(* Log/debug/error message fifo *)
FUNCTION_BLOCK FB_LogFifo
VAR_INPUT
	bLog		: BOOL 		:= FALSE;(* TRUE => Enable log message output, FALSE => Disable *)
	sPrefix		: STRING 	:= 'Unknown::';(* Log message description string (allows the identification of log message source) *)
	
	sMessage	: STRING 	:= '';(* String message to add (write) to the fifo *)
	nErrID		: UDINT 	:= 0;(* Error code to add (write) to the fifo *)
	hSocket		: T_HSOCKET;(* Socket connection handle *)
END_VAR
VAR_OUTPUT
	bOk			: BOOL;(* TRUE = New entry added or removed succesfully, FALSE = Fifo overflow or fifo empty *)
	sGet		: T_MaxString := '';(* String entry removed (read) from fifo *)
	nCount		: UDINT := 0;(* Number of fifo entries *)
END_VAR
VAR
	fbBuffer 	: FB_StringRingBuffer;(* Basic (lower level) string buffer control function block *)
	buffer		: ARRAY[0..PLCPRJ_BUFFER_SIZE] OF BYTE;(* Internal buffer memory *)
	sSource		: T_MaxString;	
	sPut		: T_MaxString;
END_VAR

;

ACTION Clear:
(* Clears all fifo entries *)
fbBuffer.A_Reset( 	pBuffer := ADR( buffer ), cbBuffer := SIZEOF( buffer ), 
					bOk=>bOk, nCount=>nCount, getValue=>sGet );
END_ACTION

ACTION Error:
(* Adds new fifo entry *)
IF nErrID = 0 THEN
	sSource := '::Error: 0x';
ELSIF ( nErrID AND 16#80000000) = 16#80000000 THEN
	IF nErrID = 16#80072746 THEN
		sSource := '::Win32 error (the connection is reset by remote side): 0x';
	ELSE
		sSource := '::Win32 error: 0x';
	END_IF
ELSIF (nErrID AND 16#00008100) = 16#00008100 THEN
	CASE nErrID OF
		PLCPRJ_ERROR_RECEIVE_TIMEOUT:
			sSource := '::PLC sample project receive timeout error: 0x';
		PLCPRJ_ERROR_SENDFIFO_OVERFLOW:
			sSource := '::PLC sample project send fifo overflow error: 0x';
		PLCPRJ_ERROR_RECFIFO_OVERFLOW:
			sSource := '::PLC sample project receive fifo overflow error: 0x';
	ELSE
		sSource := '::Other PLC sample project error: 0x';
	END_CASE
ELSIF (nErrID AND 16#00008000) = 16#00008000 THEN
	sSource := '::Internal TCP/IP Connection Server error: 0x';
ELSE
	sSource := '::TwinCAT System error: 0x';
END_IF

sPut := CONCAT( CONCAT( CONCAT( sPrefix, sMessage ), sSource ), DWORD_TO_HEXSTR( nErrID AND 16#FFFF, 0, FALSE ) ); 

fbBuffer.A_AddTail( pBuffer:= ADR(buffer), cbBuffer:= SIZEOF(buffer),
					putValue:= sPut, bOk=>bOk, nCount=>nCount );
IF bOk THEN
	IF bLog THEN(* Log error message *)
		ADSLOGSTR( ADSLOG_MSGTYPE_ERROR OR ADSLOG_MSGTYPE_LOG, '%s', sPut );	
	END_IF
END_IF
END_ACTION

ACTION Message:
(* Adds new fifo entry *)
sPut := CONCAT( CONCAT( sPrefix, sMessage ), CONCAT( '::', HSOCKET_TO_STRING(hSocket) ) );
fbBuffer.A_AddTail( pBuffer:= ADR(buffer), cbBuffer:= SIZEOF(buffer),
					putValue:= sPut, bOk=>bOk, nCount=>nCount );
IF bOk THEN
	IF bLog THEN(* Log information message *)
		ADSLOGSTR( ADSLOG_MSGTYPE_HINT OR ADSLOG_MSGTYPE_LOG, '%s', sPut );	
	END_IF
END_IF
END_ACTION

ACTION Remove:
(* Removes oldest fifo entry *)
IF nCount = 0 THEN
	sGet := '';
	bOk := FALSE;
	RETURN;
END_IF

fbBuffer.A_RemoveHead( pBuffer:= ADR(buffer), cbBuffer:= SIZEOF(buffer),
						getValue=>sGet, bOk=>bOk, nCount=>nCount );
END_ACTION

END_FUNCTION_BLOCK

(* stored: Version 1.1.0.1, ProductVersion 3.1.4024.12
   POU FB_LogFifo: Id {cf9e956c-1b38-487d-9fc5-7a973b1bb83f}, SpecialFunc None
   Action Clear: Id {02270425-d2ec-45e7-b278-aab16cb13ed5}
   Action Error: Id {4b1d4906-35e3-4161-aaf9-49e28507d240}
   Action Message: Id {a03e1481-d5bd-4918-9b4e-dc42575596f4}
   Action Remove: Id {6bbf46bc-351d-4dcc-91d2-dbfbc016f526} *)
